// TIA Portal V20 export
// export: Created 2025-12-01T14:56:27.9696857Z, ExportSetting None, DisplayName Totally Integrated Automation Portal, DisplayVersion V20 Update 3, DisplayName TIA Portal Openness, DisplayVersion V20 Update 3, DisplayName TIA Portal Version Control Interface, DisplayVersion V20 Update 3, DisplayName STEP 7 Professional, DisplayVersion V20 Update 3, DisplayName STEP 7 Safety, DisplayVersion V20 Update 2, DisplayName WinCC Basic/Comfort/Advanced, DisplayVersion V20 Update 3, DisplayName WinCC Professional, DisplayVersion V20 Update 3, DisplayName WinCC Unified, DisplayVersion V20 Update 3
ORGANIZATION_BLOCK "OB30_Interrupcion_Diag_profinet_ASi"   // OB30, LAD, CyclicInterrupt
{ S7_Optimized_Access := 'TRUE' }
// stored: SetENOAutomatically false
   VAR_INPUT
      Initial_Call : Bool;   // Initial call of this OB
      Event_Count : Int;   // Events discarded
   END_VAR
BEGIN

REGION Network 1: Diagnostico Red Profinet
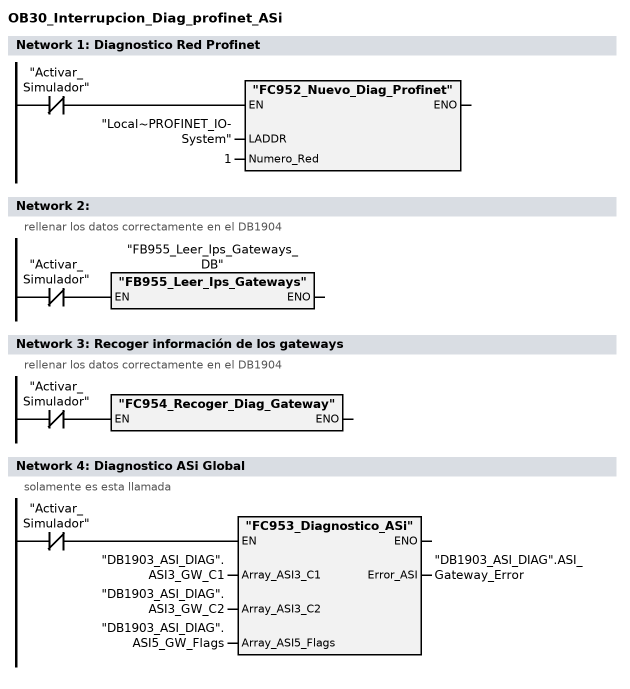
   RUNG wire#powerrail
      I_Contact( "Activar_Simulador" )
      "FC952_Nuevo_Diag_Profinet"(LADDR := "Local~PROFINET_IO-System", Numero_Red := 1)
   END_RUNG
   // the same network as SCL:
   IF NOT "Activar_Simulador" THEN
       "FC952_Nuevo_Diag_Profinet"(LADDR := "Local~PROFINET_IO-System", Numero_Red := 1);
   END_IF;
END_REGION

REGION Network 2
   // rellenar los datos correctamente en el DB1904
   RUNG wire#powerrail
      I_Contact( "Activar_Simulador" )
      "FB955_Leer_Ips_Gateways_DB"()
   END_RUNG
   // the same network as SCL:
   IF NOT "Activar_Simulador" THEN
       "FB955_Leer_Ips_Gateways_DB"();   // "FB955_Leer_Ips_Gateways"
   END_IF;
END_REGION

REGION Network 3: Recoger información de los gateways
   // rellenar los datos correctamente en el DB1904
   RUNG wire#powerrail
      I_Contact( "Activar_Simulador" )
      "FC954_Recoger_Diag_Gateway"()
   END_RUNG
   // the same network as SCL:
   IF NOT "Activar_Simulador" THEN "FC954_Recoger_Diag_Gateway"(); END_IF;
END_REGION

REGION Network 4: Diagnostico ASi Global
   // solamente es esta llamada
   RUNG wire#powerrail
      I_Contact( "Activar_Simulador" )
      "FC953_Diagnostico_ASi"(Array_ASI3_C1 := "DB1903_ASI_DIAG".ASI3_GW_C1, Array_ASI3_C2 := "DB1903_ASI_DIAG".ASI3_GW_C2, Array_ASI5_Flags := "DB1903_ASI_DIAG".ASI5_GW_Flags, Error_ASI => "DB1903_ASI_DIAG".ASI_Gateway_Error)
   END_RUNG
   // the same network as SCL:
   IF NOT "Activar_Simulador" THEN
       "FC953_Diagnostico_ASi"(Array_ASI3_C1 := "DB1903_ASI_DIAG".ASI3_GW_C1,
                               Array_ASI3_C2 := "DB1903_ASI_DIAG".ASI3_GW_C2,
                               Array_ASI5_Flags := "DB1903_ASI_DIAG".ASI5_GW_Flags,
                               Error_ASI => "DB1903_ASI_DIAG".ASI_Gateway_Error);
   END_IF;
END_REGION
END_ORGANIZATION_BLOCK
